FUNCTION_BLOCK FbInputMap
VAR
	xInput: BOOL;
	xA: BOOL;
	xB: BOOL;
END_VAR

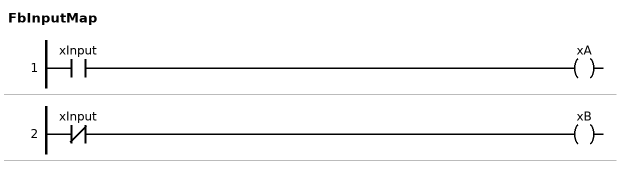
// NETWORK 1
xA := xInput;

// NETWORK 2
xB := NOT xInput;

END_FUNCTION_BLOCK

(* stored: Version 1.1.0.1, ProductVersion 3.1.4024.12
   POU FbInputMap: Id {a6ecb96f-a23e-4e30-8fd6-06e203e46085}, SpecialFunc None *)
